FUNCTION_BLOCK PresenceSensor IMPLEMENTS ITF_BinarySensor
VAR_INPUT
END_VAR
VAR_OUTPUT
END_VAR
VAR
	DI_WPDetected AT %I* : BOOL;
END_VAR

PROPERTY Value : BOOL
GET
Value := DI_WPDetected;
END_GET
END_PROPERTY

END_FUNCTION_BLOCK

(* stored: Version 1.1.0.1
   POU PresenceSensor: Id {039d7bd4-c895-40bd-ba33-10799c5c0e0b}, SpecialFunc None
   Property Value: Id {aa68a283-aca6-41bc-9f2a-8889c368dbcd}
   Get Get: Id {b5182475-fa72-45c9-97ac-ccb0e379c68b} *)
